(* CODESYS project LD_TEST.xml

Project tree, tasks and I/O mapping:
  program LD_TEST [LD]
*)

// LD_TEST
PROGRAM LD_TEST
VAR
	Sensor1: BOOL;
	Sensor2: BOOL;
	sensor3: BOOL;
	PowerOn: BOOL;
	TON_0: TON;
	CTU_0: CTU;
	PowerOff: BOOL;
	edgetrigger: BOOL;
	answer: UINT;
	BLINK_0: BLINK;
END_VAR
VAR // added by the converter: edge detectors and wires of the graphical bodies
    _rt1, _rt2 : R_TRIG;
    _w1 : BOOL;
END_VAR

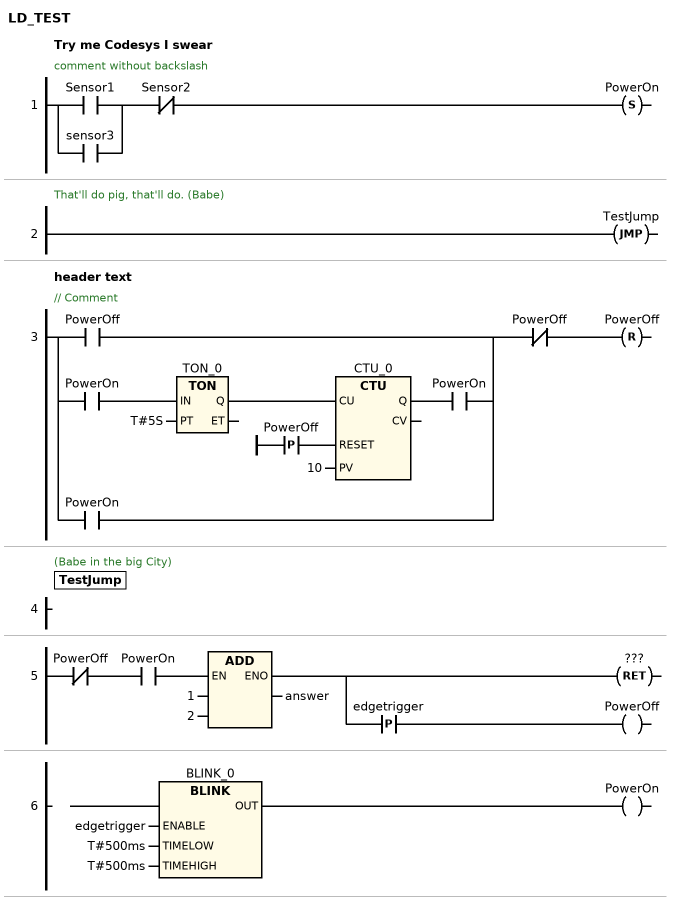
// NETWORK 1: Try me Codesys I swear
// comment without backslash
PowerOn S= (Sensor1 OR sensor3) AND NOT Sensor2;

// NETWORK 2
// That'll do pig, that'll do. (Babe)
JMP TestJump;

// NETWORK 3: header text
// // Comment
TON_0(IN := PowerOn, PT := T#5S); // TON
_rt1(CLK := PowerOff);
CTU_0(CU := TON_0.Q, RESET := _rt1.Q, PV := 10); // CTU
PowerOff R= (PowerOff OR CTU_0.Q AND PowerOn OR PowerOn) AND NOT PowerOff;

// NETWORK 4
// (Babe in the big City)
TestJump: ;

// NETWORK 5
_w1 := NOT PowerOff AND PowerOn;
IF _w1 THEN answer := 1 + 2; END_IF
IF _w1 THEN RETURN; END_IF
_rt2(CLK := edgetrigger);
PowerOff := _w1 AND _rt2.Q;

// NETWORK 6
BLINK_0(ENABLE := edgetrigger, TIMELOW := T#500ms, TIMEHIGH := T#500ms); // BLINK
PowerOn := BLINK_0.OUT;

END_PROGRAM
